// TIA Portal V21 export
VAR_GLOBAL   // PLC tag table "InputDigitali"
END_VAR
